// TIA Portal V19 export
FUNCTION "STEP_TIMER" : Void   // FC213, STL
TITLE = STEP TIMING FOR SEQUENCER
{ S7_Optimized_Access := 'TRUE' }
AUTHOR : HGS
FAMILY : Sequence
NAME : SEQ_ST
// ********************************************************************************
//                         SEQUENCE STEP TIMER
// ********************************************************************************
// 
// The sequence provides a time count for a currently active sequence step. The
// time accumulation is stored as a double-integer in the sequence data area.
// 
// The time accumulation is reset to zero when the sequence steps to the next step.
// 
// The time accumulation is the no. of "TIME_PULSE" occurrences (1-shots) that 
// have 
// happened while the particular sequence step has been active.
// 
// 
// 
// REVISION RECORD ****************************************************************
// 
// Ver   DATE      CHANGES
// 0.1   23/02/01  Under development for P851
// 0.2   26/02/01  Avoidance of time increment on reset - added as "JU end"
// stored: AutoNumber false
   VAR_INPUT
      DBNR : Int;   // Sequence Data Block Number
      NEXT_STEP_LOCATION : Int;   // Data block address of next step register
      STEP_NUM_LOCATION : Int;   // Data block address of current step register
      TIME_PULSE : Bool;   // 1-second time pulse
      STEP_TIME_ACC_LOCATION : Int;   // Data block address of step time accumulator
   END_VAR
   VAR_TEMP
      DBNR_TEMP : Int;   // Temporary integer register
      STEP_NUM_PTR : DInt;   // Address of current step number
      NEXT_STEP_PTR : DInt;   // Address of next step number
      STEP_TIME_ACC_PTR : DInt;   // Address of step time accumulator
   END_VAR
BEGIN

NETWORK
TITLE = DETECT SEQUENCE STEP TRANSITION TO ZERO THE SEQUENCE STEP TIMING
      L     #DBNR;
      T     #DBNR_TEMP;
      OPN   DB [#DBNR_TEMP];  // Reference the sequence DB
      L     #STEP_NUM_LOCATION;
      ITD;
      SLD   3;
      T     #STEP_NUM_PTR;  //  location of current step no.

      L     #NEXT_STEP_LOCATION;
      ITD;
      SLD   3;
      T     #NEXT_STEP_PTR;  //  location of next step no.

      L     #STEP_TIME_ACC_LOCATION;
      ITD;
      SLD   3;
      T     #STEP_TIME_ACC_PTR;  //  location of step time accumulator

      L     DBW [#STEP_NUM_PTR];  // current step no.
      L     DBW [#NEXT_STEP_PTR];  // next step no.
      ==I;
      JC    ichk;
      L     0;
      T     DBD [#STEP_TIME_ACC_PTR];  // Step time accumulation
      JU    end;  // Avoid time pulse check
ichk: NOP   0;



NETWORK
TITLE = CHECK TO UPDATE SEQUENCE STEP TIMING ACCUMULATOR
      AN    #TIME_PULSE;
      JC    end;
      L     DBD [#STEP_TIME_ACC_PTR];  // Step time accumulation
      L     1;
      +D;  // Increment the time count
      T     DBD [#STEP_TIME_ACC_PTR];  // and restore the time accumulation
end:  SAVE;  // "SAVE" to set BR status bit

END_FUNCTION
